///EL6900 | TwinSAFE PLC
FUNCTION_BLOCK EL6900_v0_00

END_FUNCTION_BLOCK

(* stored: Version 1.1.0.1, ProductVersion 3.1.4022.6
   POU EL6900_v0_00: Id {f88fd9c8-623c-4763-990b-4dbc24d5502f}, SpecialFunc None *)
